(* IEC 61131-3 sources: plc_benchmarking/ladder_logic_progrs/FLOPS_fixed_n/build, 2 files *)

(* ---- plc.st ---- *)
TYPE
  LOGLEVEL : (CRITICAL, WARNING, INFO, DEBUG) := INFO;
END_TYPE

FUNCTION_BLOCK LOGGER
  VAR_INPUT
    TRIG : BOOL;
    MSG : STRING;
    LEVEL : LOGLEVEL := INFO;
  END_VAR
  VAR
    TRIG0 : BOOL;
  END_VAR

  IF TRIG AND NOT TRIG0 THEN
  {{
   LogMessage(GetFbVar(LEVEL),(char*)GetFbVar(MSG, .body),GetFbVar(MSG, .len));
  }}
  END_IF;
  TRIG0:=TRIG;
END_FUNCTION_BLOCK

PROGRAM FLOPS
  VAR
    count : DINT := 0;
    num_ops : DINT := 200;
    product : REAL := 1.0;
    run_flag : BOOL := true;
    reset : BOOL := true;
    run_status : BOOL := false;
  END_VAR
  VAR
    _TMP_MUL2_ENO : BOOL;
    _TMP_MUL2_OUT : REAL;
    _TMP_SUB7_ENO : BOOL;
    _TMP_SUB7_OUT : DINT;
    _TMP_GT12_ENO : BOOL;
    _TMP_GT12_OUT : BOOL;
    _TMP_MOVE15_ENO : BOOL;
    _TMP_MOVE15_OUT : REAL;
    _TMP_LE18_ENO : BOOL;
    _TMP_LE18_OUT : BOOL;
    _TMP_MOVE28_ENO : BOOL;
    _TMP_MOVE28_OUT : DINT;
  END_VAR

  _TMP_MUL2_OUT := MUL(EN := run_flag, IN1 := product, IN2 := 5.0, ENO => _TMP_MUL2_ENO);
  IF _TMP_MUL2_ENO THEN
      product := _TMP_MUL2_OUT;
  END_IF;
  _TMP_SUB7_OUT := SUB(EN := _TMP_MUL2_ENO, IN1 := count, IN2 := 1, ENO => _TMP_SUB7_ENO);
  IF _TMP_SUB7_ENO THEN
      count := _TMP_SUB7_OUT;
  END_IF;
  _TMP_GT12_OUT := GT(EN := run_flag, IN1 := product, IN2 := 5000.0, ENO => _TMP_GT12_ENO);
  _TMP_MOVE15_OUT := MOVE(EN := _TMP_GT12_OUT, IN := 1.0, ENO => _TMP_MOVE15_ENO);
  IF _TMP_MOVE15_ENO THEN
      product := _TMP_MOVE15_OUT;
  END_IF;
  _TMP_LE18_OUT := LE(EN := run_flag, IN1 := count, IN2 := 0, ENO => _TMP_LE18_ENO);
  IF _TMP_LE18_OUT THEN
    run_flag := FALSE; (*reset*)
  END_IF;
  _TMP_MOVE28_OUT := MOVE(EN := NOT(run_flag) AND reset, IN := num_ops, ENO => _TMP_MOVE28_ENO);
  IF _TMP_MOVE28_ENO THEN
      count := _TMP_MOVE28_OUT;
  END_IF;
  IF _TMP_MOVE28_ENO THEN
    reset := FALSE; (*reset*)
  END_IF;
  run_status := _TMP_SUB7_ENO;
  IF _TMP_LE18_OUT THEN
    run_status := FALSE; (*reset*)
  END_IF;
END_PROGRAM

CONFIGURATION Config0

  RESOURCE Res0 ON PLC
    TASK task0(INTERVAL := T#20ms,PRIORITY := 0);
    PROGRAM instance0 WITH task0 : FLOPS;
  END_RESOURCE
END_CONFIGURATION

(* ---- generated_plc.st ---- *)
PROGRAM FLOPS
  VAR
    count AT %MD0 : DINT := 0;
    num_ops AT %MD1 : DINT := 200;
    product AT %MD2 : REAL := 1.0;
    run_flag AT %IX0.0 : BOOL := true;
    reset AT %IX0.1 : BOOL := true;
    run_status AT %QX0.0 : BOOL := false;
  END_VAR
  VAR
    _TMP_MUL2_ENO : BOOL;
    _TMP_MUL2_OUT : REAL;
    _TMP_SUB7_ENO : BOOL;
    _TMP_SUB7_OUT : DINT;
    _TMP_GT12_ENO : BOOL;
    _TMP_GT12_OUT : BOOL;
    _TMP_MOVE15_ENO : BOOL;
    _TMP_MOVE15_OUT : REAL;
    _TMP_LE18_ENO : BOOL;
    _TMP_LE18_OUT : BOOL;
    _TMP_MOVE28_ENO : BOOL;
    _TMP_MOVE28_OUT : DINT;
  END_VAR

  _TMP_MUL2_OUT := MUL(EN := run_flag, IN1 := product, IN2 := 5.0, ENO => _TMP_MUL2_ENO);
  IF _TMP_MUL2_ENO THEN
      product := _TMP_MUL2_OUT;
  END_IF;
  _TMP_SUB7_OUT := SUB(EN := _TMP_MUL2_ENO, IN1 := count, IN2 := 1, ENO => _TMP_SUB7_ENO);
  IF _TMP_SUB7_ENO THEN
      count := _TMP_SUB7_OUT;
  END_IF;
  _TMP_GT12_OUT := GT(EN := run_flag, IN1 := product, IN2 := 5000.0, ENO => _TMP_GT12_ENO);
  _TMP_MOVE15_OUT := MOVE(EN := _TMP_GT12_OUT, IN := 1.0, ENO => _TMP_MOVE15_ENO);
  IF _TMP_MOVE15_ENO THEN
      product := _TMP_MOVE15_OUT;
  END_IF;
  _TMP_LE18_OUT := LE(EN := run_flag, IN1 := count, IN2 := 0, ENO => _TMP_LE18_ENO);
  IF _TMP_LE18_OUT THEN
    run_flag := FALSE; (*reset*)
  END_IF;
  _TMP_MOVE28_OUT := MOVE(EN := NOT(run_flag) AND reset, IN := num_ops, ENO => _TMP_MOVE28_ENO);
  IF _TMP_MOVE28_ENO THEN
      count := _TMP_MOVE28_OUT;
  END_IF;
  IF _TMP_MOVE28_ENO THEN
    reset := FALSE; (*reset*)
  END_IF;
  run_status := _TMP_SUB7_ENO;
  IF _TMP_LE18_OUT THEN
    run_status := FALSE; (*reset*)
  END_IF;
END_PROGRAM

CONFIGURATION Config0

  RESOURCE Res0 ON PLC
    TASK task0(INTERVAL := T#20ms,PRIORITY := 0);
    PROGRAM instance0 WITH task0 : FLOPS;
  END_RESOURCE
END_CONFIGURATION
